(* Logix 5000 project; controller LeakTestAuto vendor 1 type 14 code 226 rev 37.11; software revision 37.01; part 11 of 15 *)
(* tags used below, declared in another part *)
   AOI_Conveyor_Seq : AOI_Sequencer_x64;
   AOI_Robot_Comms : AOI_CommStatus;
   AOI_RobotPos : AOI_RobotPositions;
   AOI_SeqSteps : AOI_StandardSeqSteps;
   Conveyor : udt_OutputStructure;
   Conveyor_Seq : udt_SequenceStructure_X64;
   ConveyorCleatSensorFault : BOOL;
   FailCount : COUNTER;
   HMI_OP220_ClearProcessFaultCounts_IND : BOOL;
   HMI_OP220_ClearProcessFaultCounts_PB : BOOL;
   Nest1Cylinder : udt_OutputStructure;
   Nest2Cylinder : udt_OutputStructure;
   ONS_RobotGripper : SINT;
   OP220 : udt_Mode;
   OP220_Disable3510 : BOOL;
   OP220_LeakTest : udt_ProcessFault;
   OP220_ProcessFaultsONS : DINT;
   OP220_Seq : udt_SequenceStructure_X64;
   RFID_Comp : AOI_RFIDCompare;
   RFID_DiagData : DINT[4];
   RFID_EntryStatus : DINT;
   RFID_ExpectedFixtureVal : SINT[5,12];
   RFID_FaultCode : DINT;
   RFID_ReceiveBuffer : SINT[8000];
   RFID_RWHPort1 : RWH_CMD;
   RFID_RWHPort2 : RWH_CMD;
   RFID_SendBuffer : SINT[8000];
   RFIDScanner : udt_OutputStructure;
   RFIDTag1Match : BOOL;
   RFIDTag2Match : BOOL;
   Robot : udt_OutputStructure;
   RobotGripper : udt_OutputStructure;
   RobotInputs : udt_EpsonInputs;
   RobotOutputs : udt_EpsonOutputs;
   TON_ConveyorCleatTimeout : TIMER;
   TON_ConvUnloadDelay : TIMER;
   TON_Cylinder1DownTimeout : TIMER;
   TON_Cylinder1UpTimeout : TIMER;
   TON_Cylinder2DownTimeout : TIMER;
   TON_Cylinder2UpTimeout : TIMER;
   TON_Nest1CylinderTimer : TIMER;
   TON_Nest2CylinderTimer : TIMER;
   TON_RobotReqRetry : TIMER;
   TON_RobotReqTimeout : TIMER;
   ConveyorPurgeCounter : DINT;   // Outfeed Coveyor Purge Counter
   Delay_TMR : TIMER[11];   // Delay Timers
   I_OP220_N3_CONVEYOR_CLEAT : ALIAS FOR Local:3:I.Pt13.Data;
   I_OP220_N3_CONVEYOR_LOAD : ALIAS FOR Local:3:I.Pt12.Data;
   I_OP220_N3_CONVEYOR_UNLOAD : ALIAS FOR Local:3:I.Pt14.Data;
   I_OP220_N3_MAIN_AIR_OK : ALIAS FOR Local:3:I.Pt07.Data;
   I_OP220_N3_NEST1_EXTEND : ALIAS FOR Local:3:I.Pt04.Data;
   I_OP220_N3_NEST1_HOME : ALIAS FOR Local:3:I.Pt03.Data;
   I_OP220_N3_NEST2_EXTEND : ALIAS FOR Local:3:I.Pt06.Data;
   I_OP220_N3_NEST2_HOME : ALIAS FOR Local:3:I.Pt05.Data;
   I_OP220_N3_REJECT_BIN_OK : ALIAS FOR Local:3:I.Pt09.Data;
   I_OP220_N4_CONVEYOR_ALARM_OK : ALIAS FOR Local:4:I.Pt03.Data;
   James_Dint : DINT;   // James Test Word
   O_OP220_N5_CONV_FWD : ALIAS FOR Local:5:O.Pt12.Data;
   O_OP220_N5_EN_CONV_ALM_RST : ALIAS FOR Local:5:O.Pt10.Data;
   O_OP220_N5_EN_GRIPPER_GRIP : ALIAS FOR Local:5:O.Pt14.Data;
   O_OP220_N5_EN_GRIPPER_UNGRIP : ALIAS FOR Local:5:O.Pt15.Data;
   O_OP220_N5_EN_NEST1_EXT : ALIAS FOR Local:5:O.Pt05.Data;
   O_OP220_N5_EN_NEST1_HOME : ALIAS FOR Local:5:O.Pt06.Data;
   O_OP220_N5_EN_NEST2_EXT : ALIAS FOR Local:5:O.Pt07.Data;
   O_OP220_N5_EN_NEST2_HOME : ALIAS FOR Local:5:O.Pt08.Data;
   Oneshot : DINT;   // Oneshots
   OP220_ConsumedFromMain : DINT[50];
   OP220_ConsumedFromMain_RobotPickupSafe : BOOL;
   PLC : AOI_PLC;
   ShiftChange : BOOL;
   ST1_Ignition_DataReady_Setup : BOOL;
   ST2_Ignition_DataReady_Setup : BOOL;
(* MainProgram, continued *)

ROUTINE R40_Robot   (* ladder *)
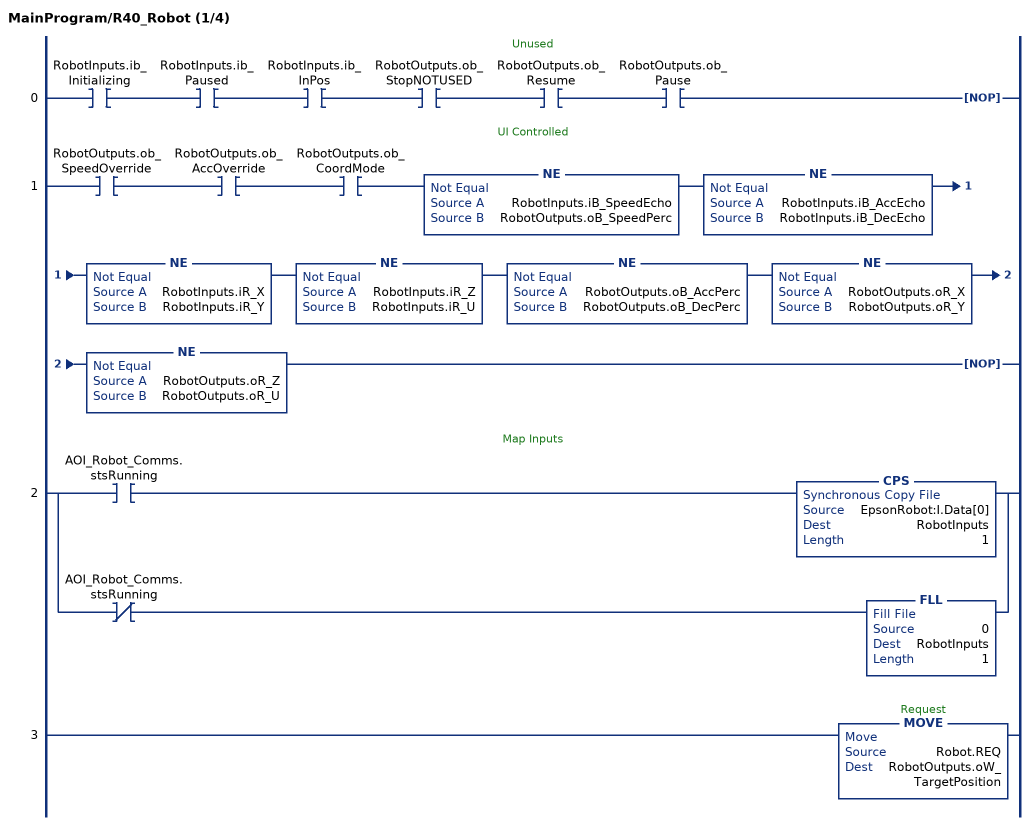
   // Unused
   0: XIC(RobotInputs.ib_Initializing)XIC(RobotInputs.ib_Paused)XIC(RobotInputs.ib_InPos)XIC(RobotOutputs.ob_StopNOTUSED)XIC(RobotOutputs.ob_Resume)XIC(RobotOutputs.ob_Pause)NOP();
   // UI Controlled
   1: XIC(RobotOutputs.ob_SpeedOverride)XIC(RobotOutputs.ob_AccOverride)XIC(RobotOutputs.ob_CoordMode)NE(RobotInputs.iB_SpeedEcho,RobotOutputs.oB_SpeedPerc)NE(RobotInputs.iB_AccEcho,RobotInputs.iB_DecEcho)NE(RobotInputs.iR_X,RobotInputs.iR_Y)NE(RobotInputs.iR_Z,RobotInputs.iR_U)NE(RobotOutputs.oB_AccPerc,RobotOutputs.oB_DecPerc)NE(RobotOutputs.oR_X,RobotOutputs.oR_Y)NE(RobotOutputs.oR_Z,RobotOutputs.oR_U)NOP();
   // Map Inputs
   2: [XIC(AOI_Robot_Comms.stsRunning) CPS(EpsonRobot:I.Data[0],RobotInputs,1) ,XIO(AOI_Robot_Comms.stsRunning) FLL(0,RobotInputs,1) ];
   3: MOVE(Robot.REQ,RobotOutputs.oW_TargetPosition);
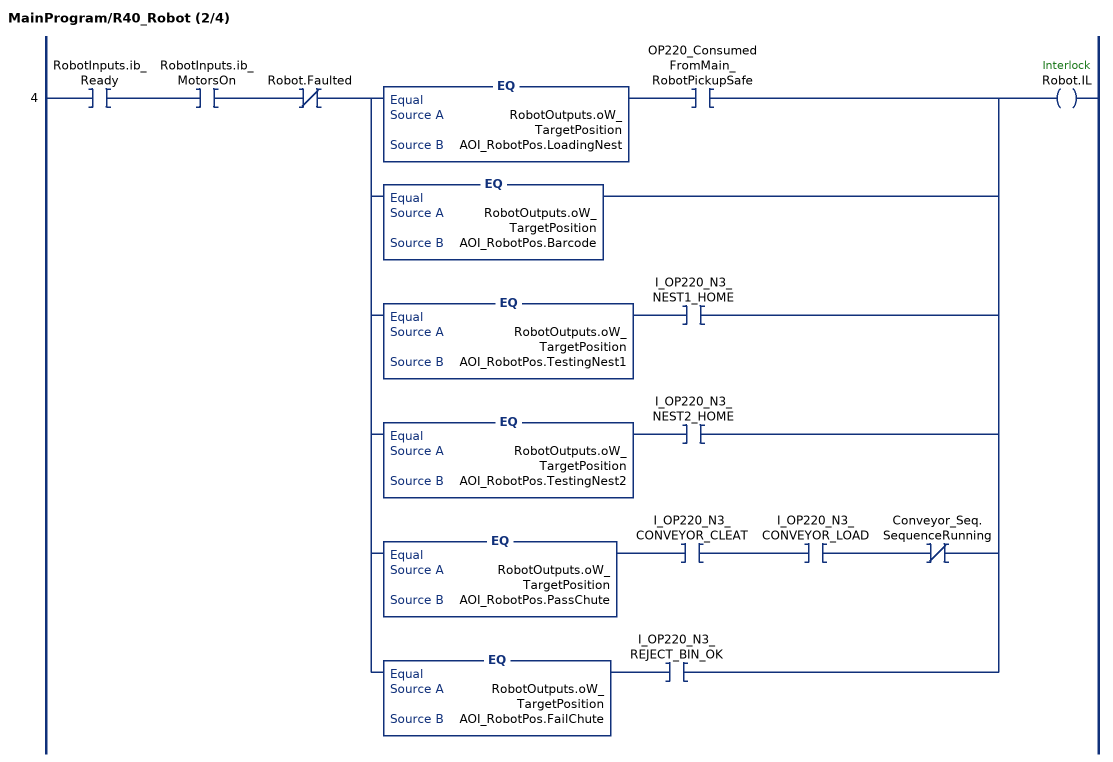
   4: XIC(RobotInputs.ib_Ready)XIC(RobotInputs.ib_MotorsOn)XIO(Robot.Faulted)[EQ(RobotOutputs.oW_TargetPosition,AOI_RobotPos.LoadingNest) XIC(OP220_ConsumedFromMain_RobotPickupSafe) ,EQ(RobotOutputs.oW_TargetPosition,AOI_RobotPos.Barcode) ,EQ(RobotOutputs.oW_TargetPosition,AOI_RobotPos.TestingNest1) XIC(I_OP220_N3_NEST1_HOME) ,EQ(RobotOutputs.oW_TargetPosition,AOI_RobotPos.TestingNest2) XIC(I_OP220_N3_NEST2_HOME) ,EQ(RobotOutputs.oW_TargetPosition,AOI_RobotPos.PassChute) XIC(I_OP220_N3_CONVEYOR_CLEAT) XIC(I_OP220_N3_CONVEYOR_LOAD) XIO(Conveyor_Seq.SequenceRunning) ,EQ(RobotOutputs.oW_TargetPosition,AOI_RobotPos.FailChute) XIC(I_OP220_N3_REJECT_BIN_OK) ]OTE(Robot.IL);
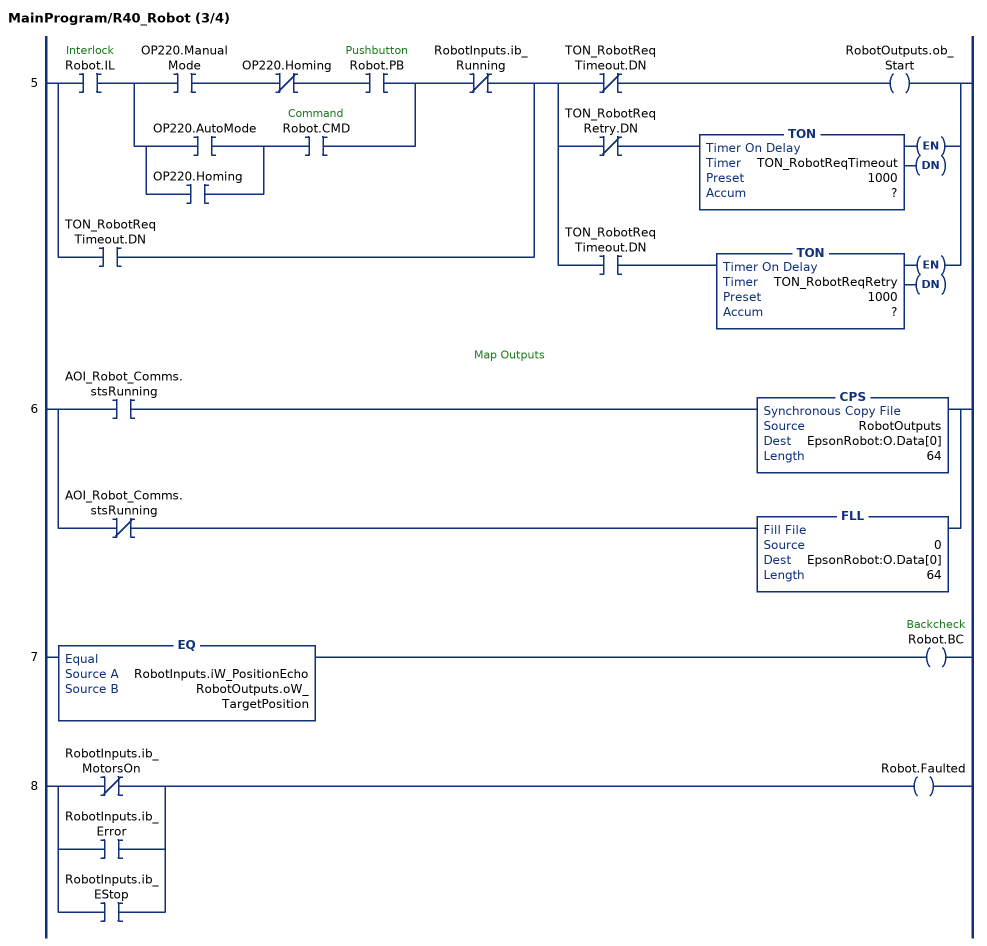
   5: [XIC(Robot.IL) [XIC(OP220.ManualMode) XIO(OP220.Homing) XIC(Robot.PB) ,[XIC(OP220.AutoMode) ,XIC(OP220.Homing) ] XIC(Robot.CMD) ] XIO(RobotInputs.ib_Running) ,XIC(TON_RobotReqTimeout.DN) ][XIO(TON_RobotReqTimeout.DN) OTE(RobotOutputs.ob_Start) ,XIO(TON_RobotReqRetry.DN) TON(TON_RobotReqTimeout,?,?) ,XIC(TON_RobotReqTimeout.DN) TON(TON_RobotReqRetry,?,?) ];
   // Map Outputs
   6: [XIC(AOI_Robot_Comms.stsRunning) CPS(RobotOutputs,EpsonRobot:O.Data[0],64) ,XIO(AOI_Robot_Comms.stsRunning) FLL(0,EpsonRobot:O.Data[0],64) ];
   7: EQ(RobotInputs.iW_PositionEcho,RobotOutputs.oW_TargetPosition)OTE(Robot.BC);
   8: [XIO(RobotInputs.ib_MotorsOn) ,XIC(RobotInputs.ib_Error) ,XIC(RobotInputs.ib_EStop) ]OTE(Robot.Faulted);
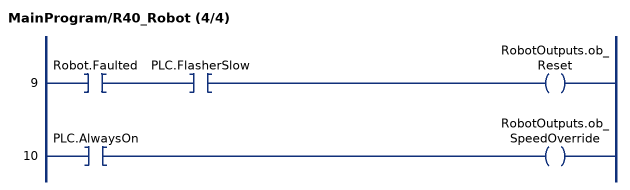
   9: XIC(Robot.Faulted)XIC(PLC.FlasherSlow)OTE(RobotOutputs.ob_Reset);
   10: XIC(PLC.AlwaysOn)OTE(RobotOutputs.ob_SpeedOverride);
END_ROUTINE

ROUTINE R41_RobotGripper   (* ladder *)
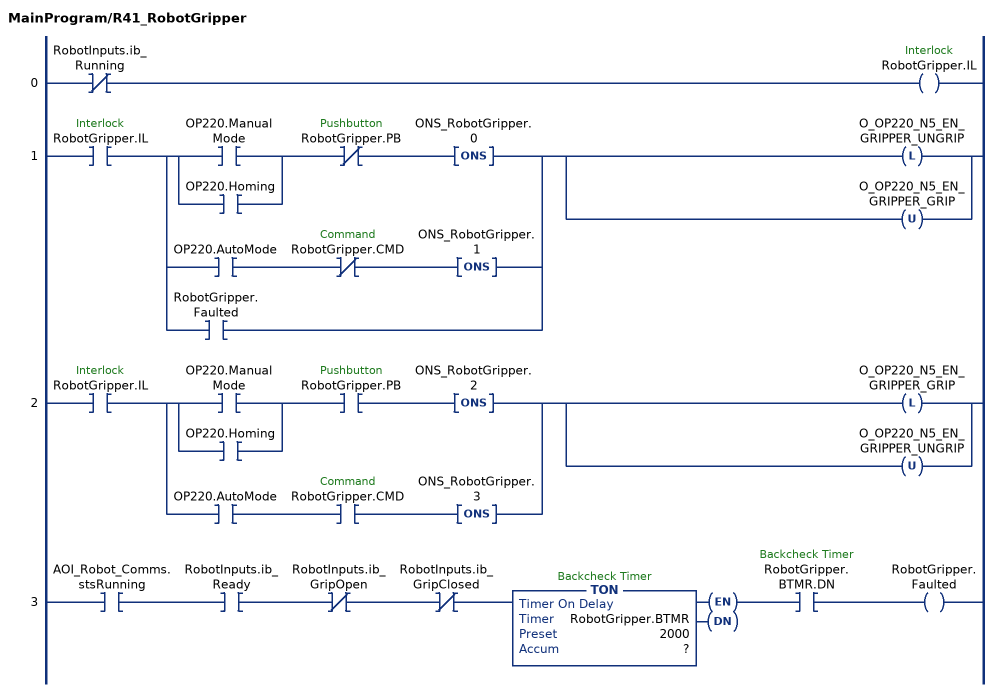
   0: XIO(RobotInputs.ib_Running)OTE(RobotGripper.IL);
   1: XIC(RobotGripper.IL)[[[XIC(OP220.ManualMode) ,XIC(OP220.Homing) ] XIO(RobotGripper.PB) ONS(ONS_RobotGripper.0) ,XIC(OP220.AutoMode) XIO(RobotGripper.CMD) ONS(ONS_RobotGripper.1) ] ,XIC(RobotGripper.Faulted) ][OTL(O_OP220_N5_EN_GRIPPER_UNGRIP) ,OTU(O_OP220_N5_EN_GRIPPER_GRIP) ];
   2: XIC(RobotGripper.IL)[[XIC(OP220.ManualMode) ,XIC(OP220.Homing) ] XIC(RobotGripper.PB) ONS(ONS_RobotGripper.2) ,XIC(OP220.AutoMode) XIC(RobotGripper.CMD) ONS(ONS_RobotGripper.3) ][OTL(O_OP220_N5_EN_GRIPPER_GRIP) ,OTU(O_OP220_N5_EN_GRIPPER_UNGRIP) ];
   3: XIC(AOI_Robot_Comms.stsRunning)XIC(RobotInputs.ib_Ready)XIO(RobotInputs.ib_GripOpen)XIO(RobotInputs.ib_GripClosed)TON(RobotGripper.BTMR,?,?)XIC(RobotGripper.BTMR.DN)OTE(RobotGripper.Faulted);
END_ROUTINE

ROUTINE R50_Conveyor   (* ladder *)
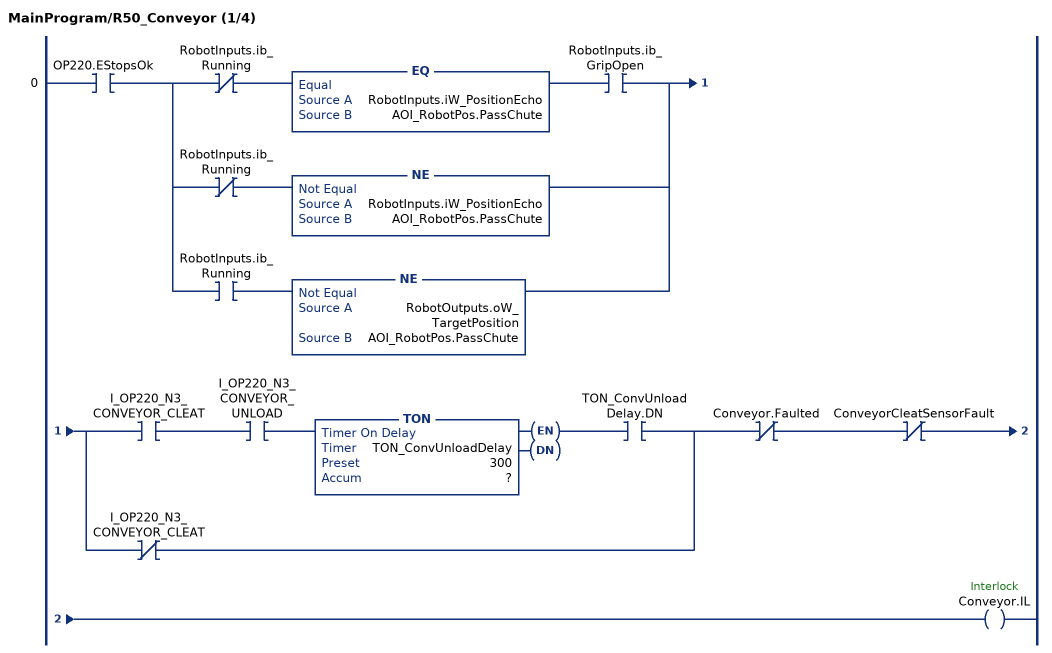
   0: XIC(OP220.EStopsOk)[XIO(RobotInputs.ib_Running) EQ(RobotInputs.iW_PositionEcho,AOI_RobotPos.PassChute) XIC(RobotInputs.ib_GripOpen) ,XIO(RobotInputs.ib_Running) NE(RobotInputs.iW_PositionEcho,AOI_RobotPos.PassChute) ,XIC(RobotInputs.ib_Running) NE(RobotOutputs.oW_TargetPosition,AOI_RobotPos.PassChute) ][XIC(I_OP220_N3_CONVEYOR_CLEAT) XIC(I_OP220_N3_CONVEYOR_UNLOAD) TON(TON_ConvUnloadDelay,?,?) XIC(TON_ConvUnloadDelay.DN) ,XIO(I_OP220_N3_CONVEYOR_CLEAT) ]XIO(Conveyor.Faulted)XIO(ConveyorCleatSensorFault)OTE(Conveyor.IL);
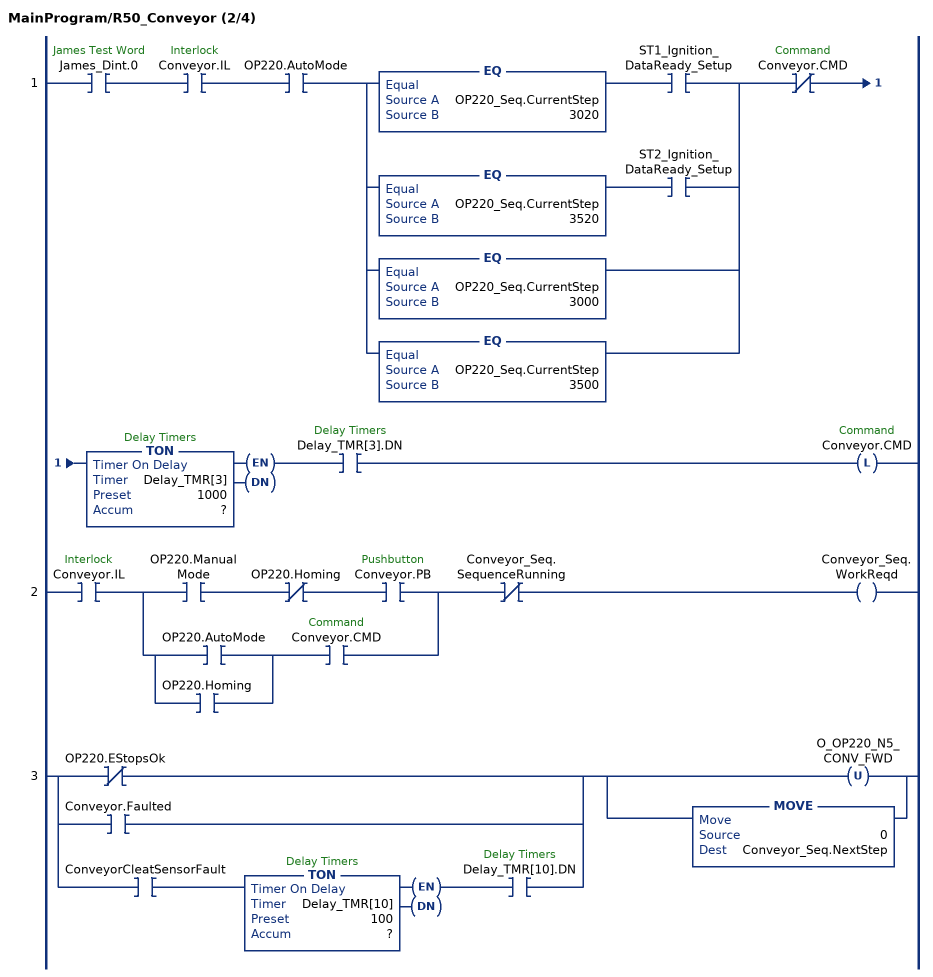
   1: XIC(James_Dint.0)XIC(Conveyor.IL)XIC(OP220.AutoMode)[EQ(OP220_Seq.CurrentStep,3020) XIC(ST1_Ignition_DataReady_Setup) ,EQ(OP220_Seq.CurrentStep,3520) XIC(ST2_Ignition_DataReady_Setup) ,EQ(OP220_Seq.CurrentStep,3000) ,EQ(OP220_Seq.CurrentStep,3500) ]XIO(Conveyor.CMD)TON(Delay_TMR[3],?,?)XIC(Delay_TMR[3].DN)OTL(Conveyor.CMD);
   2: XIC(Conveyor.IL)[XIC(OP220.ManualMode) XIO(OP220.Homing) XIC(Conveyor.PB) ,[XIC(OP220.AutoMode) ,XIC(OP220.Homing) ] XIC(Conveyor.CMD) ]XIO(Conveyor_Seq.SequenceRunning)OTE(Conveyor_Seq.WorkReqd);
   3: [XIO(OP220.EStopsOk) ,XIC(Conveyor.Faulted) ,XIC(ConveyorCleatSensorFault) TON(Delay_TMR[10],?,?) XIC(Delay_TMR[10].DN) ][OTU(O_OP220_N5_CONV_FWD) ,MOVE(0,Conveyor_Seq.NextStep) ];
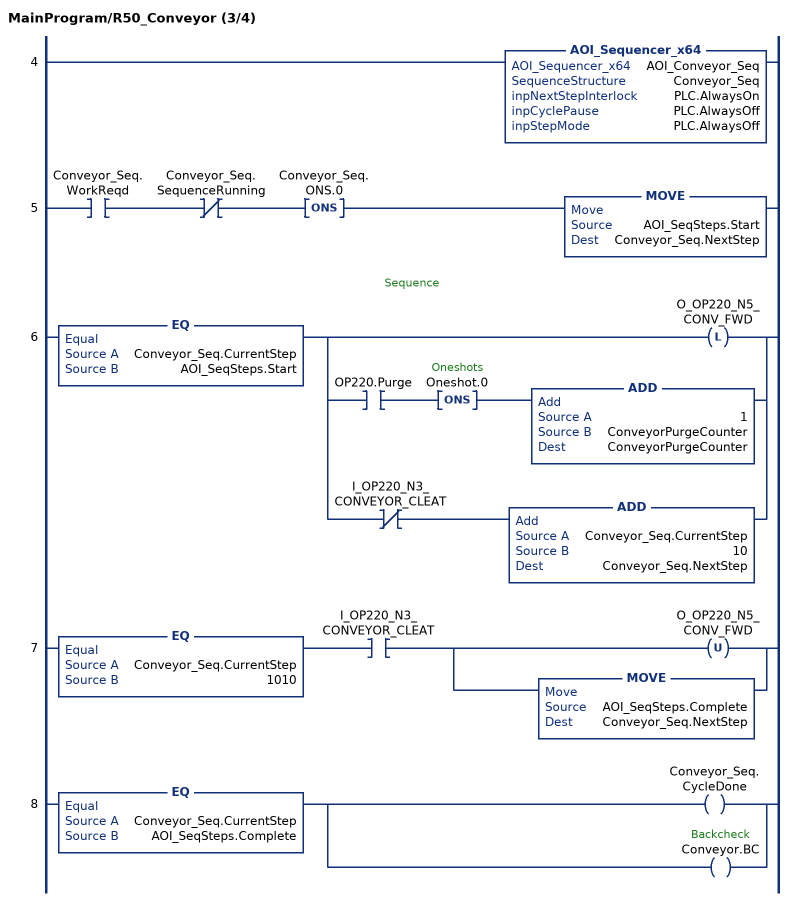
   4: AOI_Sequencer_x64(AOI_Conveyor_Seq,Conveyor_Seq,PLC.AlwaysOn,PLC.AlwaysOff,PLC.AlwaysOff);
   5: XIC(Conveyor_Seq.WorkReqd)XIO(Conveyor_Seq.SequenceRunning)ONS(Conveyor_Seq.ONS.0)MOVE(AOI_SeqSteps.Start,Conveyor_Seq.NextStep);
   // Sequence
   6: EQ(Conveyor_Seq.CurrentStep,AOI_SeqSteps.Start)[OTL(O_OP220_N5_CONV_FWD) ,XIC(OP220.Purge) ONS(Oneshot.0) ADD(1,ConveyorPurgeCounter,ConveyorPurgeCounter) ,XIO(I_OP220_N3_CONVEYOR_CLEAT) ADD(Conveyor_Seq.CurrentStep,10,Conveyor_Seq.NextStep) ];
   7: EQ(Conveyor_Seq.CurrentStep,1010)XIC(I_OP220_N3_CONVEYOR_CLEAT)[OTU(O_OP220_N5_CONV_FWD) ,MOVE(AOI_SeqSteps.Complete,Conveyor_Seq.NextStep) ];
   8: EQ(Conveyor_Seq.CurrentStep,AOI_SeqSteps.Complete)[OTE(Conveyor_Seq.CycleDone) ,OTE(Conveyor.BC) ];
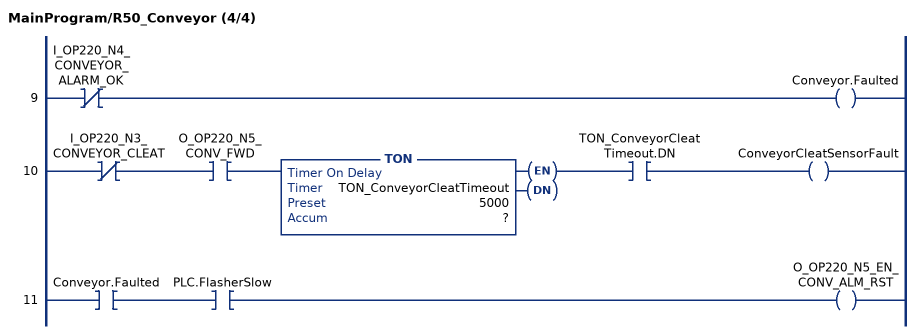
   9: XIO(I_OP220_N4_CONVEYOR_ALARM_OK)OTE(Conveyor.Faulted);
   10: XIO(I_OP220_N3_CONVEYOR_CLEAT)XIC(O_OP220_N5_CONV_FWD)TON(TON_ConveyorCleatTimeout,?,?)XIC(TON_ConveyorCleatTimeout.DN)OTE(ConveyorCleatSensorFault);
   11: XIC(Conveyor.Faulted)XIC(PLC.FlasherSlow)OTE(O_OP220_N5_EN_CONV_ALM_RST);
END_ROUTINE

ROUTINE R60_Nest1Cylinder   (* ladder *)
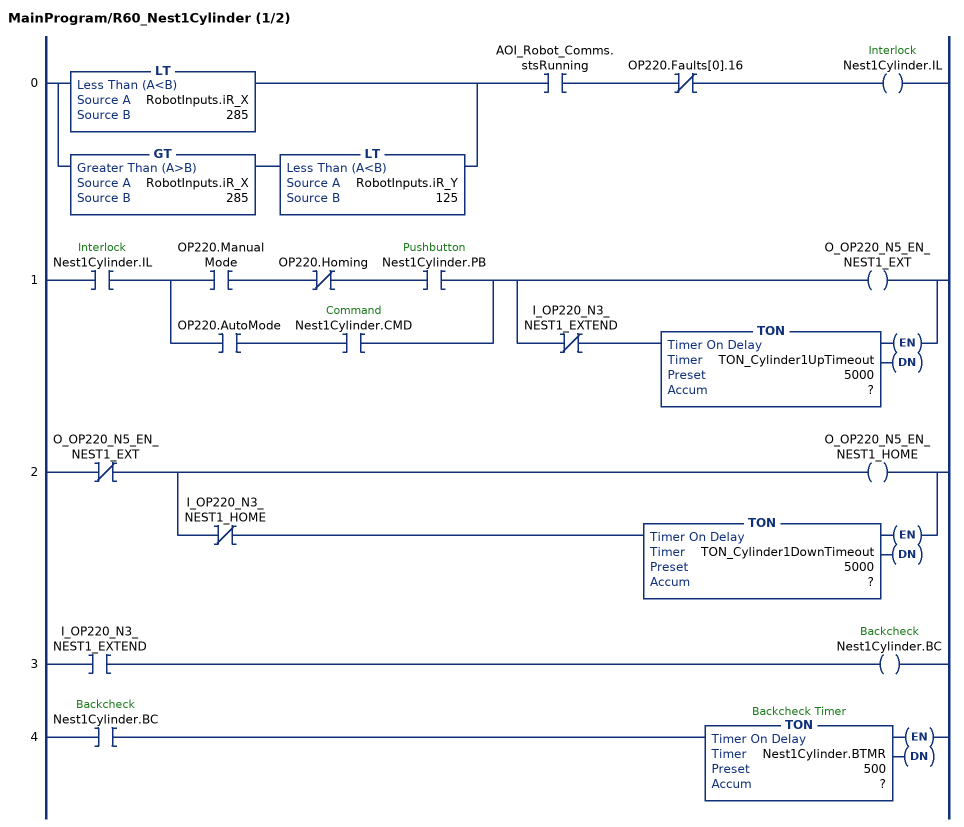
   0: [LT(RobotInputs.iR_X,285) ,GT(RobotInputs.iR_X,285) LT(RobotInputs.iR_Y,125) ]XIC(AOI_Robot_Comms.stsRunning)XIO(OP220.Faults[0].16)OTE(Nest1Cylinder.IL);
   1: XIC(Nest1Cylinder.IL)[XIC(OP220.ManualMode) XIO(OP220.Homing) XIC(Nest1Cylinder.PB) ,XIC(OP220.AutoMode) XIC(Nest1Cylinder.CMD) ][OTE(O_OP220_N5_EN_NEST1_EXT) ,XIO(I_OP220_N3_NEST1_EXTEND) TON(TON_Cylinder1UpTimeout,?,?) ];
   2: XIO(O_OP220_N5_EN_NEST1_EXT)[OTE(O_OP220_N5_EN_NEST1_HOME) ,XIO(I_OP220_N3_NEST1_HOME) TON(TON_Cylinder1DownTimeout,?,?) ];
   3: XIC(I_OP220_N3_NEST1_EXTEND)OTE(Nest1Cylinder.BC);
   4: XIC(Nest1Cylinder.BC)TON(Nest1Cylinder.BTMR,?,?);
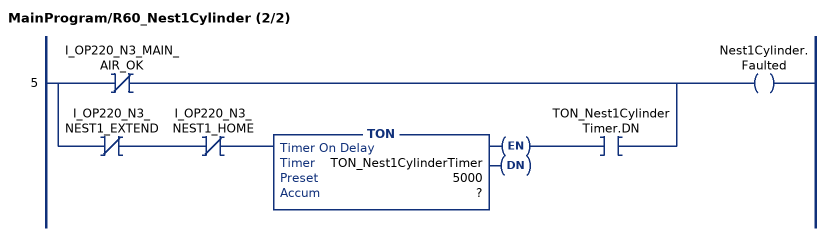
   5: [XIO(I_OP220_N3_MAIN_AIR_OK) ,XIO(I_OP220_N3_NEST1_EXTEND) XIO(I_OP220_N3_NEST1_HOME) TON(TON_Nest1CylinderTimer,?,?) XIC(TON_Nest1CylinderTimer.DN) ]OTE(Nest1Cylinder.Faulted);
END_ROUTINE

ROUTINE R61_Nest2Cylinder   (* ladder *)
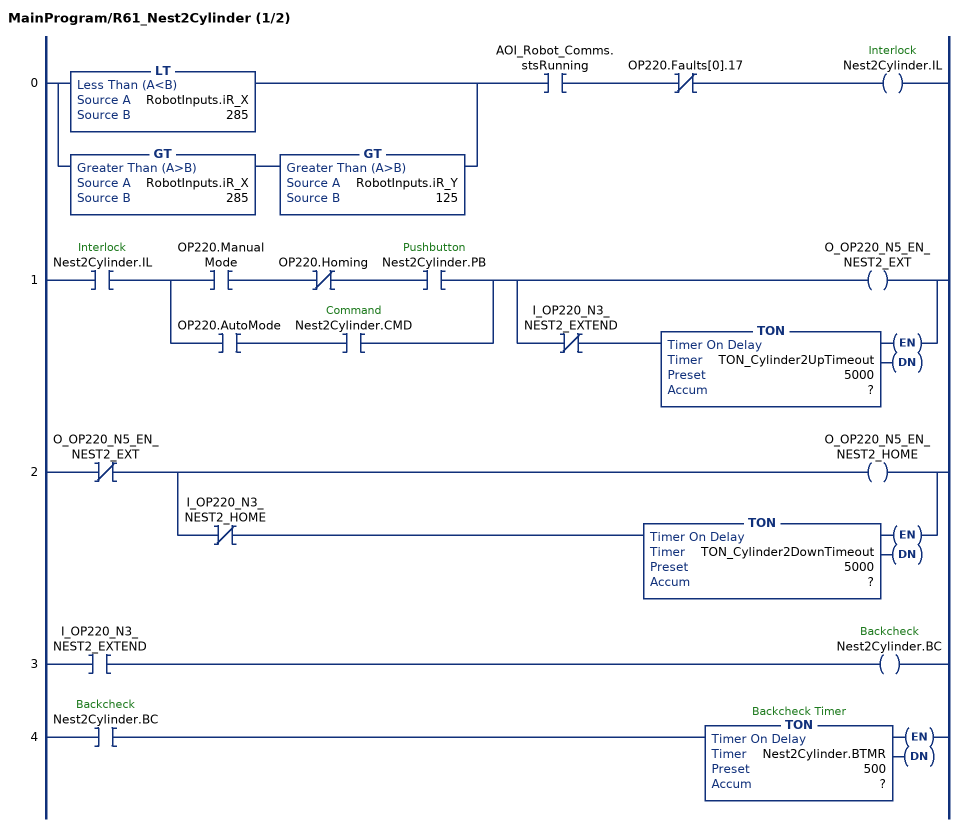
   0: [LT(RobotInputs.iR_X,285) ,GT(RobotInputs.iR_X,285) GT(RobotInputs.iR_Y,125) ]XIC(AOI_Robot_Comms.stsRunning)XIO(OP220.Faults[0].17)OTE(Nest2Cylinder.IL);
   1: XIC(Nest2Cylinder.IL)[XIC(OP220.ManualMode) XIO(OP220.Homing) XIC(Nest2Cylinder.PB) ,XIC(OP220.AutoMode) XIC(Nest2Cylinder.CMD) ][OTE(O_OP220_N5_EN_NEST2_EXT) ,XIO(I_OP220_N3_NEST2_EXTEND) TON(TON_Cylinder2UpTimeout,?,?) ];
   2: XIO(O_OP220_N5_EN_NEST2_EXT)[OTE(O_OP220_N5_EN_NEST2_HOME) ,XIO(I_OP220_N3_NEST2_HOME) TON(TON_Cylinder2DownTimeout,?,?) ];
   3: XIC(I_OP220_N3_NEST2_EXTEND)OTE(Nest2Cylinder.BC);
   4: XIC(Nest2Cylinder.BC)TON(Nest2Cylinder.BTMR,?,?);
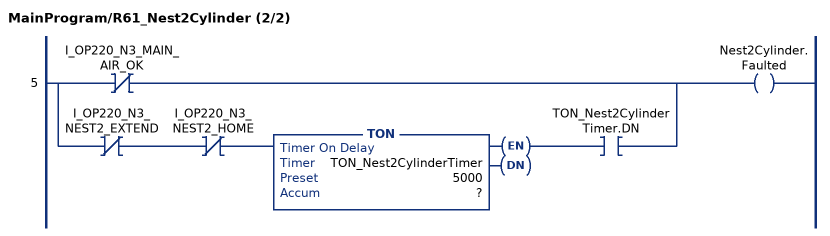
   5: [XIO(I_OP220_N3_MAIN_AIR_OK) ,XIO(I_OP220_N3_NEST2_EXTEND) XIO(I_OP220_N3_NEST2_HOME) TON(TON_Nest2CylinderTimer,?,?) XIC(TON_Nest2CylinderTimer.DN) ]OTE(Nest2Cylinder.Faulted);
END_ROUTINE

ROUTINE R70_RFID   (* ladder *)
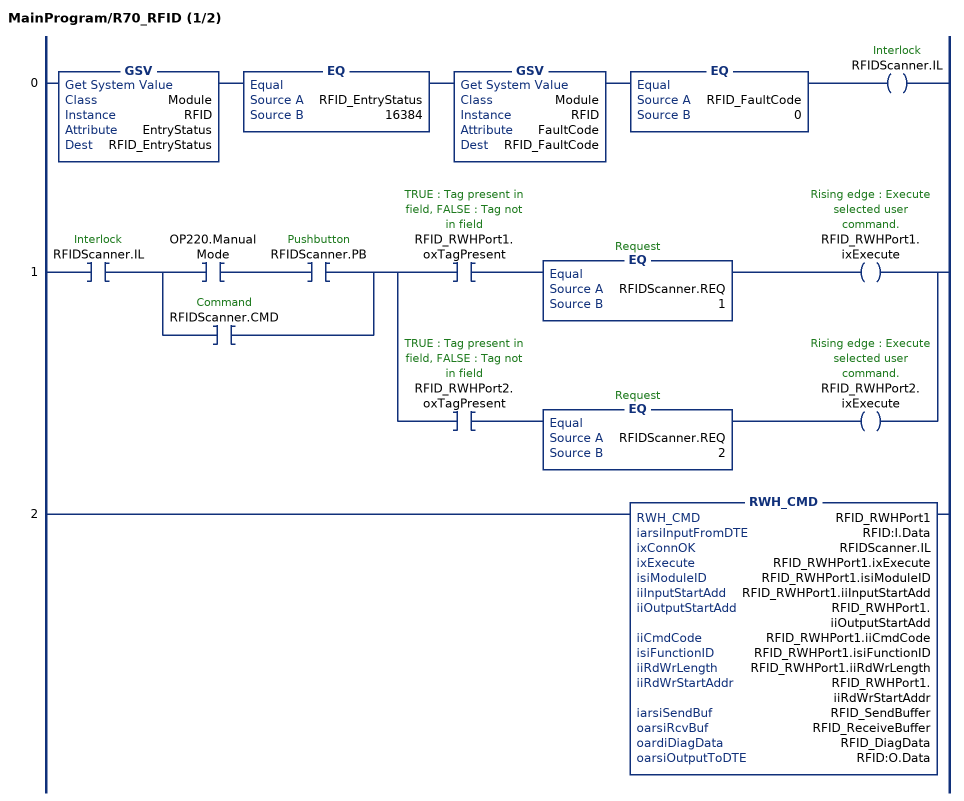
   0: GSV(Module,RFID,EntryStatus,RFID_EntryStatus)EQ(RFID_EntryStatus,16384)GSV(Module,RFID,FaultCode,RFID_FaultCode)EQ(RFID_FaultCode,0)OTE(RFIDScanner.IL);
   1: XIC(RFIDScanner.IL)[XIC(OP220.ManualMode) XIC(RFIDScanner.PB) ,XIC(RFIDScanner.CMD) ][XIC(RFID_RWHPort1.oxTagPresent) EQ(RFIDScanner.REQ,1) OTE(RFID_RWHPort1.ixExecute) ,XIC(RFID_RWHPort2.oxTagPresent) EQ(RFIDScanner.REQ,2) OTE(RFID_RWHPort2.ixExecute) ];
   2: RWH_CMD(RFID_RWHPort1,RFID:I.Data,RFIDScanner.IL,RFID_RWHPort1.ixExecute,RFID_RWHPort1.isiModuleID,RFID_RWHPort1.iiInputStartAdd,RFID_RWHPort1.iiOutputStartAdd,RFID_RWHPort1.iiCmdCode,RFID_RWHPort1.isiFunctionID,RFID_RWHPort1.iiRdWrLength,RFID_RWHPort1.iiRdWrStartAddr,RFID_SendBuffer,RFID_ReceiveBuffer,RFID_DiagData,RFID:O.Data);
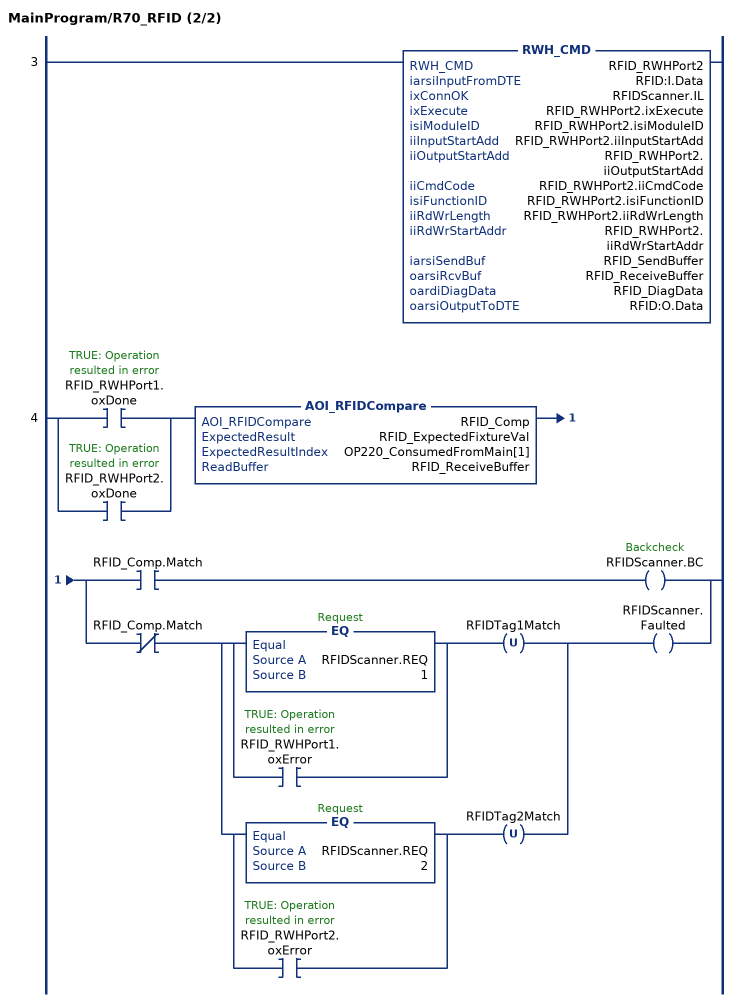
   3: RWH_CMD(RFID_RWHPort2,RFID:I.Data,RFIDScanner.IL,RFID_RWHPort2.ixExecute,RFID_RWHPort2.isiModuleID,RFID_RWHPort2.iiInputStartAdd,RFID_RWHPort2.iiOutputStartAdd,RFID_RWHPort2.iiCmdCode,RFID_RWHPort2.isiFunctionID,RFID_RWHPort2.iiRdWrLength,RFID_RWHPort2.iiRdWrStartAddr,RFID_SendBuffer,RFID_ReceiveBuffer,RFID_DiagData,RFID:O.Data);
   4: [XIC(RFID_RWHPort1.oxDone) ,XIC(RFID_RWHPort2.oxDone) ]AOI_RFIDCompare(RFID_Comp,RFID_ExpectedFixtureVal,OP220_ConsumedFromMain[1],RFID_ReceiveBuffer)[XIC(RFID_Comp.Match) OTE(RFIDScanner.BC) ,XIO(RFID_Comp.Match) [[EQ(RFIDScanner.REQ,1) ,XIC(RFID_RWHPort1.oxError) ] OTU(RFIDTag1Match) ,[EQ(RFIDScanner.REQ,2) ,XIC(RFID_RWHPort2.oxError) ] OTU(RFIDTag2Match) ] OTE(RFIDScanner.Faulted) ];
END_ROUTINE

ROUTINE R89_3_5_10_Alarms   (* ladder *)
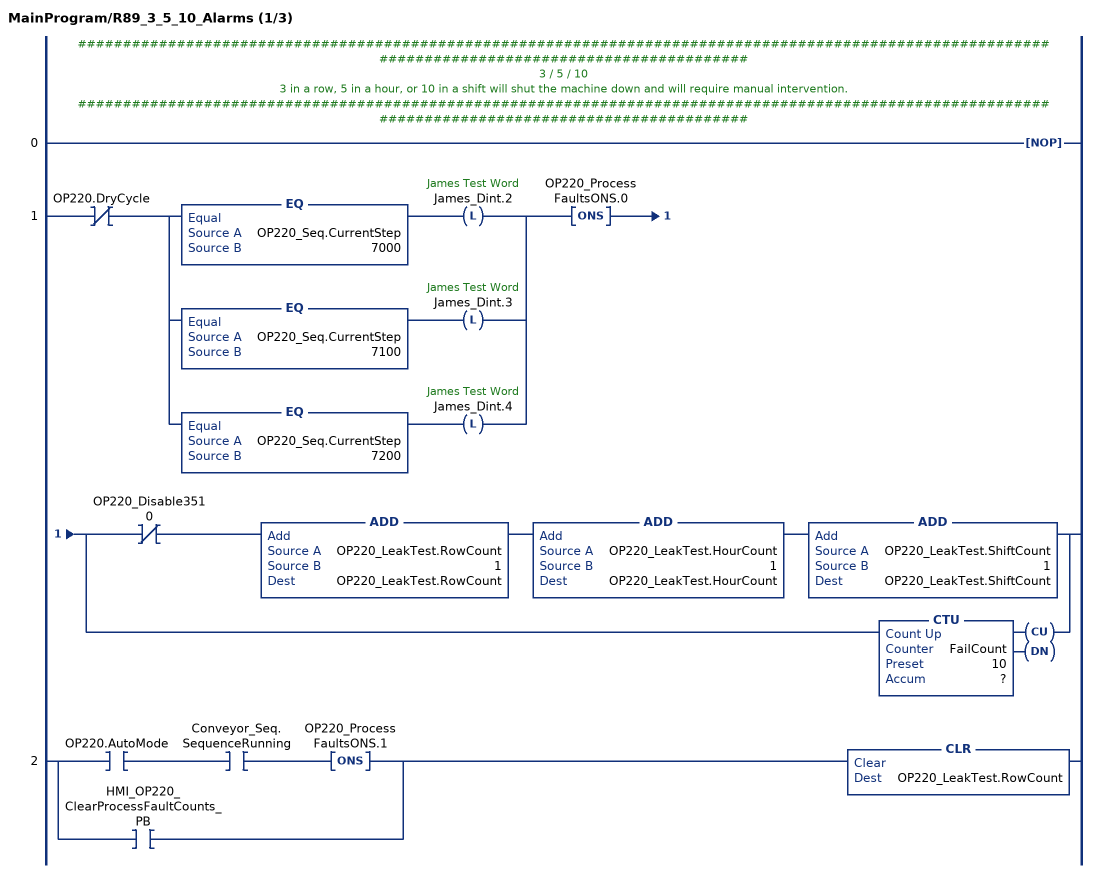
   // #####################################################################################################################################################
   // 3 / 5 / 10
   // 	3 in a row, 5 in a hour, or 10 in a shift will shut the machine down and will require manual intervention.
   // #####################################################################################################################################################
   0: NOP();
   1: XIO(OP220.DryCycle)[EQ(OP220_Seq.CurrentStep,7000) OTL(James_Dint.2) ,EQ(OP220_Seq.CurrentStep,7100) OTL(James_Dint.3) ,EQ(OP220_Seq.CurrentStep,7200) OTL(James_Dint.4) ]ONS(OP220_ProcessFaultsONS.0)[XIO(OP220_Disable3510) ADD(OP220_LeakTest.RowCount,1,OP220_LeakTest.RowCount) ADD(OP220_LeakTest.HourCount,1,OP220_LeakTest.HourCount) ADD(OP220_LeakTest.ShiftCount,1,OP220_LeakTest.ShiftCount) ,CTU(FailCount,?,?) ];
   2: [XIC(OP220.AutoMode) XIC(Conveyor_Seq.SequenceRunning) ONS(OP220_ProcessFaultsONS.1) ,XIC(HMI_OP220_ClearProcessFaultCounts_PB) ]CLR(OP220_LeakTest.RowCount);
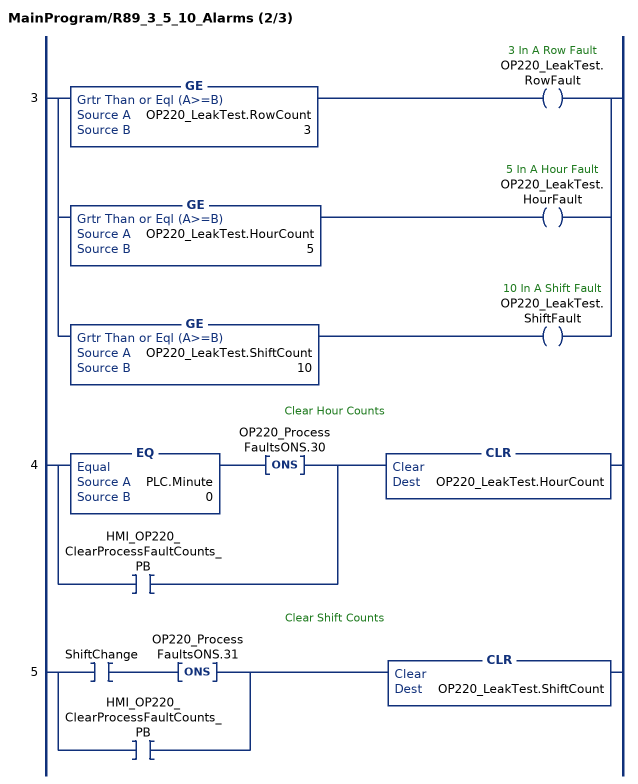
   3: [GE(OP220_LeakTest.RowCount,3) OTE(OP220_LeakTest.RowFault) ,GE(OP220_LeakTest.HourCount,5) OTE(OP220_LeakTest.HourFault) ,GE(OP220_LeakTest.ShiftCount,10) OTE(OP220_LeakTest.ShiftFault) ];
   // Clear Hour Counts
   4: [EQ(PLC.Minute,0) ONS(OP220_ProcessFaultsONS.30) ,XIC(HMI_OP220_ClearProcessFaultCounts_PB) ]CLR(OP220_LeakTest.HourCount);
   // Clear Shift Counts
   5: [XIC(ShiftChange) ONS(OP220_ProcessFaultsONS.31) ,XIC(HMI_OP220_ClearProcessFaultCounts_PB) ]CLR(OP220_LeakTest.ShiftCount);
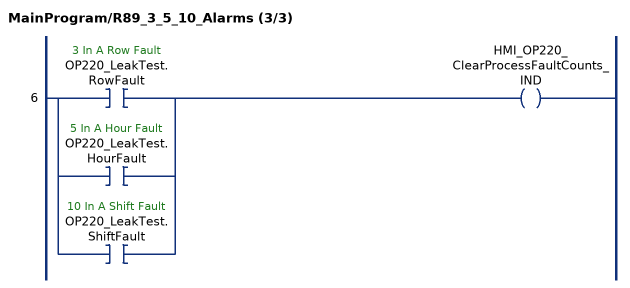
   6: [XIC(OP220_LeakTest.RowFault) ,XIC(OP220_LeakTest.HourFault) ,XIC(OP220_LeakTest.ShiftFault) ]OTE(HMI_OP220_ClearProcessFaultCounts_IND);
END_ROUTINE
